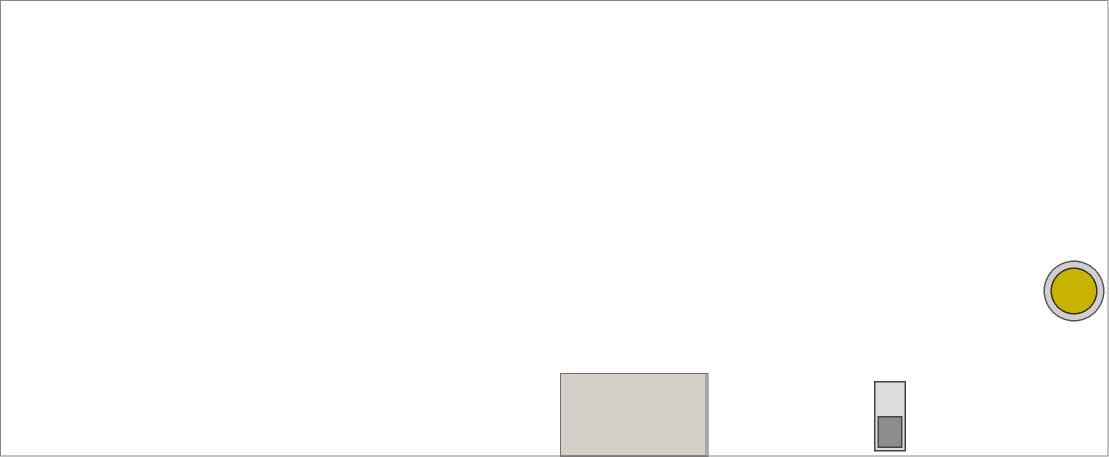
VISUALIZATION Visualization  // 1109x457
    Button (560,373 148x84)
    DipSwitch (855,381 70x70), variable: MAIN.bTimerIn, behaviour: TOGGLE, style: Switch-DipSwitch-Gray
    Lamp1 (1039,256 70x70), variable: MAIN.bTimerEnded, style: Lamp-Lamp1-Yellow
END_VISUALIZATION

(* stored: Version 1.1.0.1, ProductVersion 3.1.4024.9
   Visu Visualization: Id {354ea08c-5554-429e-934a-20077cb5c671} *)
